(* PLC project Tc2_System.FB_EOF Demo, tc3-libraries-kb TwinCAT 3.1 *)
(* stored: creationDateTime 2026-05-20T00:00:00, modificationDateTime 2026-05-20T00:00:00 *)

PROGRAM P_Demo_FB_EOF
  VAR
    fbEof : FB_EOF;  (* FB_EOF 实例 *)
    hOpenedFile : UINT;  (* 已打开句柄 *)
    bEofCheckRequest : BOOL;  (* 在线写 TRUE 触发一次查询 *)
    bEofReached : BOOL;  (* TRUE = 已到 EOF *)
    bEofError : BOOL;  (* TRUE = 查询失败 *)
    nErrIdLast : UDINT;  (* ADS 错误号 *)
    bBusyMon : BOOL;  (* ADS 通讯中 *)
  END_VAR

// =============================================================================
// 场景：按块循环读完整个大日志文件，每读完一块就显式查询是否到达 EOF 作为退出条件。
// 价值：语义比 FB_FileRead 内置 bEOF 更清晰，专做检测。
// 验证：读到中间时 bEofReached = FALSE；读到末尾 → bEofReached = TRUE。
// 验证步骤：
//   1. 右键 PLC 项目 → Import PLCopenXML → 选本文件
//   2. 引用 Tc2_System（References → Add library）
//   3. 编译 → 登录 → 运行；按上方『验证』行的指示在线写值观察
// =============================================================================

fbEof(
    sNetId   := '',
    hFile    := hOpenedFile,
    bExecute := bEofCheckRequest,
    tTimeout := T#10S,
    bBusy    => bBusyMon,
    bError   => bEofError,
    nErrId   => nErrIdLast,
    bEOF     => bEofReached
);
END_PROGRAM
